// TIA Portal V19 export
DATA_BLOCK "Config"   // DB135
// stored: Access Published, MemoryReserve 100, Namespace Unit2.Em6
   VAR
      em { ExternalWritable := 'False'} : "LAF_typeEmConfiguration";   // Configuration of EM Parameters
      em6Parameters : "LAF_typePlasticRollerEm6Parameters";
   END_VAR
BEGIN
   em.referenceDesignator.parent := WSTRING#'U1';
   em.referenceDesignator.relative := WSTRING#'EM1';
END_DATA_BLOCK
